PROGRAM AnalogConversion_obs
VAR
	i					: INT := 1; //charger 1-6
	j					: INT := 1;  // section 1 - 4 
	k					: INT := 1;  // cap 1-10
	m					: INT := 1; //form cap 1-12
END_VAR

//MCP Charger 
//Analog Input
FOR i := 1 TO 6 BY 1 DO 
	//MCP_IO.Charger[i].voltageSP := (HMI_DB.TDKLoad[i].RequiredChargedV *1000);
	MCP_IO.Charger[i].voltageSP := (1000*Setpoints.TDKLoad[i].RequiredChargedV);
END_FOR

//charger 1 is 30kV *************************************************************************************
MCP_IO.Charger[1].voltageFeedback_norm := Norm_x (raw_input := INT_TO_REAL (MCP_IO.Charger[1].voltageFeedback_raw),
														x_max := 32767,
														x_min := 0);
MCP_IO.Charger[1].voltageFeedback := (30000 - 0) * ADC_10V(normal_input := MCP_IO.Charger[1].voltageFeedback_norm,
															x_max := 10,
															x_min := 0);
															
	MCP_IO.Charger[1].currentFeedback_norm := Norm_x (raw_input := INT_TO_REAL (MCP_IO.Charger[1].currentFeedback_raw),
														x_max := 32767,
														x_min := 0);
	// 30kV charger max current output is 0.6A													
	MCP_IO.Charger[1].currentFeedback := (0.6 - 0) * ADC_10V(normal_input := MCP_IO.Charger[1].currentFeedback_norm,
															x_max := 10,
															x_min := 0);																							
//*************************************************************************************

FOR i := 2 TO 6 BY 1 DO
	
	MCP_IO.Charger[i].ChargerType_12kV := NOT MCP_IO.Charger[i].ChargerType_50kV;
	//voltage
	MCP_IO.Charger[i].voltageFeedback_norm := Norm_x (raw_input := INT_TO_REAL (MCP_IO.Charger[i].voltageFeedback_raw),
														x_max := 32767,
														x_min := 0);
	//current																									
	MCP_IO.Charger[i].currentFeedback_norm := Norm_x (raw_input := INT_TO_REAL (MCP_IO.Charger[i].currentFeedback_raw),
														x_max := 32767,
														x_min := 0);
	//50kV chargers feedback
	//if 50kV config selected
	IF MCP_IO.Charger[i].ChargerType_50kV = TRUE THEN 
		//50kv
		MCP_IO.Charger[i].voltageFeedback := (EngVal.Max_50kVChargerVoltage - EngVal.Min_50kVChargerVoltage) * ADC_10V(
																							normal_input := MCP_IO.Charger[i].voltageFeedback_norm,
																							x_max := 10,
																							x_min := 0);

		MCP_IO.Charger[i].currentFeedback := (EngVal.Max_50kVChargerCurrent - EngVal.Min_50kVChargerCurrent) * ADC_10V(
																							normal_input := MCP_IO.Charger[i].currentFeedback_norm,
																							x_max := 10,
																							x_min := 0);
		//12kv
	ELSIF MCP_IO.Charger[i].ChargerType_12kV = TRUE THEN
		MCP_IO.Charger[i].voltageFeedback := (EngVal.Max_12kVChargerVoltage - EngVal.Min_12kVChargerVoltage) * ADC_10V(normal_input := MCP_IO.Charger[i].voltageFeedback_norm,
																														x_max := 10,
																														x_min := 0);
		MCP_IO.Charger[i].currentFeedback := (EngVal.Max_12kVChargerCurrent - EngVal.Min_12kVChargerCurrent) * ADC_10V(
																							normal_input := MCP_IO.Charger[i].currentFeedback_norm,
																							x_max := 10,
																							x_min := 0);										
	END_IF;	
END_FOR;

//Analog Output
//voltageSP = Required Charge Voltage**
//limit for charing the cap

//Charger 1 is 30kV *************************************
IF MCP_IO.Charger[1].voltageSP >= (12000) THEN
			MCP_IO.Charger[1].voltageSP := 10000; //limit at 35kV
		ELSIF MCP_IO.Charger[1].voltageSP <= 0 THEN
			MCP_IO.Charger[1].voltageSP := 0; //limit at 0V
		END_IF; 

//prepare output signal for 30kV chargers.  //**Setpoints.RequiredChargedV -> MCP_IO.Charger.voltageSP **
MCP_IO.Charger[1].voltageSP_norm := Norm_x (raw_input := (MCP_IO.Charger[1].voltageSP), 
												x_max := 30000,
												x_min := 0);
		
MCP_IO.Charger[1].voltageSP_raw := AQ (norm_input := MCP_IO.Charger[1].voltageSP_norm, 
												x_max := 10,
												x_min := 0); 
	
												
//limite for output sigal (<= 10V)  this should not happen
IF MCP_IO.Charger[1].voltageSP_raw >= 32767 THEN 
	MCP_IO.Charger[1].voltageSP_raw := 32767; 										
END_IF;
//*******************************************************

//FOR i := 1 TO 8 BY 1 DO
FOR i := 2 TO 6 BY 1 DO	
	
	//if 50kV config selected
	IF MCP_IO.Charger[i].ChargerType_50kV = TRUE THEN 
		//set limits of charger voltage input 
		IF MCP_IO.Charger[i].voltageSP >= (EngVal.UpperLimit50kVCaps) THEN
			MCP_IO.Charger[i].voltageSP := 35000; //limit at 35kV
		ELSIF MCP_IO.Charger[i].voltageSP <= 0 THEN
			MCP_IO.Charger[i].voltageSP := 0; //limit at 0V
		END_IF; 
		
		(*//set limites of charger voltage input from HMI input
		IF 1000*(Setpoints.TDKLoad[i].RequiredChargedV) >= EngVal.UpperLimit50kVCaps THEN
			Setpoints.TDKLoad[i].RequiredChargedV := (EngVal.UpperLimit50kVCaps/1000); //limit at 35kv
		ELSIF Setpoints.TDKLoad[i].RequiredChargedV <= 0 THEN
			Setpoints.TDKLoad[i].RequiredChargedV :=0 ;
		END_IF*)
		
	//prepare output signal for 50kV chargers.
		MCP_IO.Charger[i].voltageSP_norm := Norm_x (raw_input :=(MCP_IO.Charger[i].voltageSP), 
												x_max := EngVal.Max_50kVChargerVoltage,
												x_min := EngVal.Min_50kVChargerVoltage);	
												
		MCP_IO.Charger[i].voltageSP_raw := AQ (norm_input := MCP_IO.Charger[i].voltageSP_norm, 
												x_max := 10,
												x_min := 0);
	END_IF;
		
	//if 12kV config selected
	IF MCP_IO.Charger[i].ChargerType_12kV = TRUE THEN
		//set limits of charger voltage input 
		IF MCP_IO.Charger[i].voltageSP <= 0 THEN
			MCP_IO.Charger[i].voltageSP := ABS(MCP_IO.Charger[i].voltageSP);
		END_IF
		
		IF MCP_IO.Charger[i].voltageSP >= (EngVal.UpperLimit12kVCaps) THEN
			MCP_IO.Charger[i].voltageSP := 10000; //limit at 10kV
		END_IF;
		
		//set limites of charger voltage input from HMI input
		(*IF 1000*(Setpoints.TDKLoad[i].RequiredChargedV) >= EngVal.UpperLimit12kVCaps THEN
			Setpoints.TDKLoad[i].RequiredChargedV := EngVal.UpperLimit12kVCaps/1000; //limit at 10kv
		ELSIF Setpoints.TDKLoad[i].RequiredChargedV <= 0 THEN
			Setpoints.TDKLoad[i].RequiredChargedV := ABS(Setpoints.TDKLoad[i].RequiredChargedV);
		END_IF
		*)
		//prepare output signal for 12kV chargers.  //**Setpoints.RequiredChargedV -> MCP_IO.Charger.voltageSP **
		MCP_IO.Charger[i].voltageSP_norm := Norm_x (raw_input := (MCP_IO.Charger[i].voltageSP), 
												x_max := EngVal.Max_12kVChargerVoltage,
												x_min := EngVal.Min_12kVChargerVoltage);
		
		MCP_IO.Charger[i].voltageSP_raw := AQ (norm_input := MCP_IO.Charger[i].voltageSP_norm, 
												x_max := 10,
												x_min := 0); 
	END_IF;	
												
	//limite for output sigal (<= 10V)  this should not happen
	IF MCP_IO.Charger[i].voltageSP_raw >= 32767 THEN 
		MCP_IO.Charger[i].voltageSP_raw := 32767; 										
	END_IF;
	
END_FOR;

//Cap voltage feedback

VoltMonitor_DB.VoltageReading_norm[0] := Norm_x (raw_input := INT_TO_REAL (VoltMonitor_DB.VoltageReading_raw[0]),
														x_max := 904, //10bit value - 1110001000 = 904deci
														x_min := 100);
LCP1_IO.Segment[1].Module[1].VoltageFeedback := (12000 - 0) * ADC_10V(normal_input := VoltMonitor_DB.VoltageReading_norm[0],
																		x_max := 10,
																		x_min := 0);														


//reset counter
//IF i > 8 THEN
IF i > 6 THEN
	i := 1;
END_IF;

IF j > 3 THEN 
	j := 1;
END_IF

IF k > 10 THEN 
	k := 1;
END_IF

IF m > 12 THEN 
	m := 1;
END_IF

END_PROGRAM

(* stored: Version 1.1.0.1, ProductVersion 3.1.4024.11
   POU AnalogConversion_obs: Id {3b8eecca-a8e5-4cfd-bb8d-8865397a6f0b}, SpecialFunc None *)
